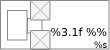
VISUALIZATION SperrAntrieb_MR_Flap_Txt_R_Below  // 110x50
VAR_INPUT
    ITF_SPERRANTRIEB_IN   	:   ITF_SPERRANTRIEB;	
END_VAR
VAR_INPUT CONSTANT
    stExklParameter		:   STRING[40] := ' ';	
END_VAR
VAR CONSTANT
	uiIconNr				:	UINT := 7;
END_VAR
    Frame (0,0 110x50), invisible if: NOT fcCheckQuerryReturnIcon(_ITF_In := ITF_SPERRANTRIEB_IN,_uiIconNr_In := uiIconNr)
        shows SperrAntrieb_MR_Flap_RB_CheckQuerry(ITF_SPERRANTRIEB_IN := ITF_SPERRANTRIEB_IN, stExklParameter := stExklParameter)
        shows Icon()
END_VISUALIZATION

// 40 Visualizations/ICON/SperrAntrieb_RIGHT/Motor_Right/Below/SperrAntrieb_MR_Flap_RB_CheckQuerry
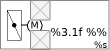
VISUALIZATION SperrAntrieb_MR_Flap_RB_CheckQuerry  // 110x50
VAR_INPUT
    ITF_SPERRANTRIEB_IN   :   ITF_SPERRANTRIEB;
    stExklParameter		:   STRING[40];	
END_VAR
    Frame (0,0 110x50)
        shows SperrAntrieb_MR_Flap_RB_CheckEnabled(ITF_SPERRANTRIEB_IN := ITF_SPERRANTRIEB_IN, stExklParameter := stExklParameter)
END_VISUALIZATION

// 40 Visualizations/ICON/SperrAntrieb_RIGHT/Motor_Right/Below/SperrAntrieb_MR_Flap_RB_CheckEnabled
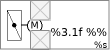
VISUALIZATION SperrAntrieb_MR_Flap_RB_CheckEnabled  // 110x50
VAR_INPUT
    ITF_SPERRANTRIEB_IN   :   ITF_SPERRANTRIEB;
    stExklParameter		:   STRING[40];	
END_VAR
    Frame (0,0 50x50), invisible if: NOT ITF_SPERRANTRIEB_IN.proIsEnabled
        shows Icon_MR_Klappe(ITF_SPERRANTRIEB_IN := ITF_SPERRANTRIEB_IN)
    Frame (50,25 60x25), invisible if: NOT ITF_SPERRANTRIEB_IN.proIsEnabled
        shows ValueDwnUp(ITF_SPERRANTRIEB_IN := ITF_SPERRANTRIEB_IN, uiTextAusrichtung := 4)
    Rectangle (0,0 110x50)
        OnMouseClick:  Dialog=SperrAntrieb_POPUP, Parameters={stExklParameter: , ITF_SPERRANTRIEBIN: ITF_SPERRANTRIEB_IN, uiPopUpGruppe: 0}, OpenCentered=True
END_VISUALIZATION

// 40 Visualizations/ICON/SperrAntrieb_BASE/Ventile/Klappe/Motor_Below/MB_Klappe_AUF
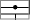
VISUALIZATION MB_Klappe_AUF  // 30x20
    Rectangle (0,0 30x14)
    Line (15,14) (15,20)
    Line (0,7) (30,7)
    Ellipse (13,5 4x4)
END_VISUALIZATION

// 40 Visualizations/ICON/SperrAntrieb_BASE/Ventile/Klappe/Motor_Left/ML_Klappe_AUF
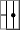
VISUALIZATION ML_Klappe_AUF  // 20x30
    Rectangle (6,0 14x30)
    Ellipse (11,13 4x4)
    Line (13,0) (13,30)
    Line (6,15) (0,15)
END_VISUALIZATION

// 40 Visualizations/ICON/SperrAntrieb_BASE/Ventile/Klappe/Motor_Right/MR_Klappe_AUF
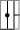
VISUALIZATION MR_Klappe_AUF  // 20x30
    Line (20,15) (14,15)
    Rectangle (0,0 14x30)
    Ellipse (5,13 4x4)
    Line (7,0) (7,30)
END_VISUALIZATION

// 40 Visualizations/ICON/SperrAntrieb_LEFT/Motor_Below/SperrAntrieb_MB_Flap_LB_CheckEnabled
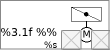
VISUALIZATION SperrAntrieb_MB_Flap_LB_CheckEnabled  // 110x50
VAR_INPUT
    ITF_SPERRANTRIEB_IN   :   ITF_SPERRANTRIEB;	
    stExklParameter		:   STRING[40];	
END_VAR
    Frame (61,0 50x50), invisible if: NOT ITF_SPERRANTRIEB_IN.proIsEnabled
        shows Icon_MB_Klappe(ITF_SPERRANTRIEB_IN := ITF_SPERRANTRIEB_IN)
    Frame (0,25 60x25), invisible if: NOT ITF_SPERRANTRIEB_IN.proIsEnabled
        shows ValueDwnUp(ITF_SPERRANTRIEB_IN := ITF_SPERRANTRIEB_IN, uiTextAusrichtung := 6)
    Rectangle (0,0 110x50)
        OnMouseClick:  Dialog=SperrAntrieb_POPUP, Parameters={stExklParameter: stExklParameter, ITF_SPERRANTRIEBIN: ITF_SPERRANTRIEB_IN, uiPopUpGruppe: 0}, OpenCentered=True
END_VISUALIZATION

// 40 Visualizations/ICON/SperrAntrieb_LEFT/Motor_Below/SperrAntrieb_MB_Flap_LB_CheckQuerry
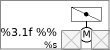
VISUALIZATION SperrAntrieb_MB_Flap_LB_CheckQuerry  // 110x50
VAR_INPUT
    ITF_SPERRANTRIEB_IN   :   ITF_SPERRANTRIEB;
    stExklParameter		:   STRING[40];	
END_VAR
    Frame (0,0 110x50)
        shows SperrAntrieb_MB_Flap_LB_CheckEnabled(ITF_SPERRANTRIEB_IN := ITF_SPERRANTRIEB_IN, stExklParameter := stExklParameter)
END_VISUALIZATION

// 40 Visualizations/ICON/SperrAntrieb_LEFT/Motor_Below/SperrAntrieb_MB_Flap_Txt_L_Below
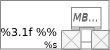
VISUALIZATION SperrAntrieb_MB_Flap_Txt_L_Below  // 110x50
VAR_INPUT
    ITF_SPERRANTRIEB_IN		:   ITF_SPERRANTRIEB;	
END_VAR
VAR_INPUT CONSTANT
    stExklParameter		:   STRING[40] := ' ';	
END_VAR
VAR CONSTANT
	uiIconNr				:	UINT := 1;
END_VAR
    Frame (0,0 110x50), invisible if: NOT fcCheckQuerryReturnIcon(_ITF_In := ITF_SPERRANTRIEB_IN,_uiIconNr_In := uiIconNr)
        shows SperrAntrieb_MB_Flap_LB_CheckQuerry(ITF_SPERRANTRIEB_IN := ITF_SPERRANTRIEB_IN, stExklParameter := stExklParameter)
        shows Icon()
END_VISUALIZATION

// 40 Visualizations/ICON/SperrAntrieb_LEFT/Motor_LEFT/Above/SperrAntrieb_ML_Flap_Txt_L_Above
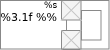
VISUALIZATION SperrAntrieb_ML_Flap_Txt_L_Above  // 110x50
VAR_INPUT
    ITF_SPERRANTRIEB_IN		:   ITF_SPERRANTRIEB;	
END_VAR
VAR_INPUT CONSTANT
    stExklParameter		:   STRING[40] := ' ';	
END_VAR
VAR CONSTANT
	uiIconNr				:	UINT := 2;
END_VAR
    Frame (0,0 110x50), invisible if: NOT fcCheckQuerryReturnIcon(_ITF_In := ITF_SPERRANTRIEB_IN,_uiIconNr_In := uiIconNr)
        shows SperrAntrieb_ML_Flap_LA_CheckQuerry(ITF_SPERRANTRIEB_IN := ITF_SPERRANTRIEB_IN, stExklParameter := stExklParameter)
        shows S_AT_ML_Valve_AB_Up_LA_CheckQuerry()
END_VISUALIZATION

// 40 Visualizations/ICON/SperrAntrieb_LEFT/Motor_LEFT/Above/SperrAntrieb_ML_Flap_LA_CheckQuerry
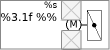
VISUALIZATION SperrAntrieb_ML_Flap_LA_CheckQuerry  // 110x50
VAR_INPUT
    ITF_SPERRANTRIEB_IN   :   ITF_SPERRANTRIEB;
    stExklParameter		:   STRING[40];	
END_VAR
    Frame (0,0 110x50)
        shows SperrAntrieb_ML_Flap_LA_CheckEnabled(ITF_SPERRANTRIEB_IN := ITF_SPERRANTRIEB_IN, stExklParameter := stExklParameter)
END_VISUALIZATION

// 40 Visualizations/ICON/SperrAntrieb_LEFT/Motor_LEFT/Above/SperrAntrieb_ML_Flap_LA_CheckEnabled
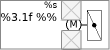
VISUALIZATION SperrAntrieb_ML_Flap_LA_CheckEnabled  // 110x50
VAR_INPUT
    ITF_SPERRANTRIEB_IN   :   ITF_SPERRANTRIEB;
    stExklParameter		:   STRING[40];	
END_VAR
    Frame (61,0 50x50), invisible if: NOT ITF_SPERRANTRIEB_IN.proIsEnabled
        shows Icon_ML_Klappe(ITF_SPERRANTRIEB_IN := ITF_SPERRANTRIEB_IN)
    Frame (0,0 60x25), invisible if: NOT ITF_SPERRANTRIEB_IN.proIsEnabled
        shows ValueUpDwn(ITF_SPERRANTRIEB_IN := ITF_SPERRANTRIEB_IN, uiTextAusrichtung := 6)
    Rectangle (0,0 110x50)
        OnMouseClick:  Dialog=SperrAntrieb_POPUP, Parameters={stExklParameter: stExklParameter, ITF_SPERRANTRIEBIN: ITF_SPERRANTRIEB_IN, uiPopUpGruppe: 0}, OpenCentered=True
END_VISUALIZATION

// 40 Visualizations/ICON/SperrAntrieb_LEFT/Motor_LEFT/Below/SperrAntrieb_ML_Flap_Txt_L_Below
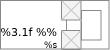
VISUALIZATION SperrAntrieb_ML_Flap_Txt_L_Below  // 110x50
VAR_INPUT
    ITF_SPERRANTRIEB_IN		:   ITF_SPERRANTRIEB;	
END_VAR
VAR_INPUT CONSTANT
    stExklParameter		:   STRING[40] := ' ';	
END_VAR
VAR CONSTANT
	uiIconNr				:	UINT := 3;
END_VAR
    Frame (0,0 110x50), invisible if: NOT fcCheckQuerryReturnIcon(_ITF_In := ITF_SPERRANTRIEB_IN,_uiIconNr_In := uiIconNr)
        shows SperrAntrieb_ML_Flap_LB_CheckQuerry(ITF_SPERRANTRIEB_IN := ITF_SPERRANTRIEB_IN, stExklParameter := stExklParameter)
        shows Icon()
END_VISUALIZATION

// 40 Visualizations/ICON/SperrAntrieb_LEFT/Motor_LEFT/Below/SperrAntrieb_ML_Flap_LB_CheckQuerry
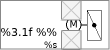
VISUALIZATION SperrAntrieb_ML_Flap_LB_CheckQuerry  // 110x50
VAR_INPUT
    ITF_SPERRANTRIEB_IN   :   ITF_SPERRANTRIEB;
    stExklParameter		:   STRING[40];	
END_VAR
    Frame (0,0 110x50)
        shows SperrAntrieb_ML_Flap_LB_CheckEnabled(ITF_SPERRANTRIEB_IN := ITF_SPERRANTRIEB_IN, stExklParameter := stExklParameter)
END_VISUALIZATION

// 40 Visualizations/ICON/SperrAntrieb_LEFT/Motor_LEFT/Below/SperrAntrieb_ML_Flap_LB_CheckEnabled
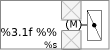
VISUALIZATION SperrAntrieb_ML_Flap_LB_CheckEnabled  // 110x50
VAR_INPUT
    ITF_SPERRANTRIEB_IN   :   ITF_SPERRANTRIEB;
    stExklParameter		:   STRING[40];	
END_VAR
    Frame (61,0 50x50), invisible if: NOT ITF_SPERRANTRIEB_IN.proIsEnabled
        shows Icon_ML_Klappe(ITF_SPERRANTRIEB_IN := ITF_SPERRANTRIEB_IN)
    Frame (0,25 60x25), invisible if: NOT ITF_SPERRANTRIEB_IN.proIsEnabled
        shows ValueDwnUp(ITF_SPERRANTRIEB_IN := ITF_SPERRANTRIEB_IN, uiTextAusrichtung := 6)
    Rectangle (0,0 110x50)
        OnMouseClick:  Dialog=SperrAntrieb_POPUP, Parameters={stExklParameter: , ITF_SPERRANTRIEBIN: ITF_SPERRANTRIEB_IN, uiPopUpGruppe: 0}, OpenCentered=True
END_VISUALIZATION

// 40 Visualizations/POPUP/PARAMETER/SperrAntrieb_Icon_SperrAntrieb
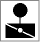
VISUALIZATION SperrAntrieb_Icon_SperrAntrieb  // 40x42
    Ellipse (13,3 14x14)
    Polygon (5,38) (5,24) (35,38)
    Polygon (5,23) (35,37) (35,23)
    Ellipse (17,27 6x6)
    Line (20,24) (20,17)
END_VISUALIZATION

// 40 Visualizations/ICON/SperrAntrieb_BASE/Value/ValueUpDwn
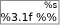
VISUALIZATION ValueUpDwn  // 60x25
VAR_INPUT
    ITF_SPERRANTRIEB_IN   :   ITF_SPERRANTRIEB;	
END_VAR
VAR_INPUT CONSTANT
    uiTextAusrichtung   : UINT := 4;    // 0 = Oben links | 1 = Horizontal zentriert | 2 = Rechts | 4 = Vertikal zentriert | 8 = Unten
END_VAR
    Textfield (0,0 60x10), "%s", text variable: ITF_SPERRANTRIEB_IN.proGetBMK, invisible if: ITF_SPERRANTRIEB_IN.proNoBmkInList
        p3718999670: uiTextAusrichtung
    Textfield (0,10 60x15), "%3.1f %%", text variable: ITF_SPERRANTRIEB_IN.proOnY, invisible if: ITF_SPERRANTRIEB_IN.proNotShowAI_ActualPosition OR NOT ITF_SPERRANTRIEB_IN.proNotShowDI_RükIsClosed OR NOT ITF_SPERRANTRIEB_IN.proNotShowDI_RükIsOpen
        p3718999670: uiTextAusrichtung
    Textfield (0,10 60x15), invisible if: NOT ITF_SPERRANTRIEB_IN.proNotShowAI_ActualPosition, text list: 'KlappenStatus', text index: ITF_SPERRANTRIEB_IN.proKlappenStatus
        p3718999670: uiTextAusrichtung
END_VISUALIZATION

// 40 Visualizations/POPUP/PARAMETER/SperrAntrieb_POPUP_IO_ITF
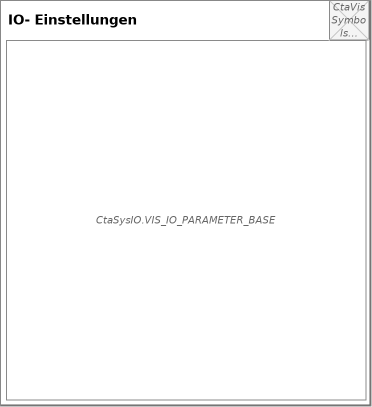
VISUALIZATION SperrAntrieb_POPUP_IO_ITF  // 372x407
VAR_INPUT
    ITF_IO_IN    :   CtaSysIO.ITF_IO;	
END_VAR
    RoundedRectangle (0,0 370x405)
    Frame (6,40 360x360)
        shows CtaSysIO.VIS_IO_PARAMETER_BASE(ITF_IO_IN := ITF_IO_IN)
        shows VIS_ANTRIEB_PARAMETER_IO1(ITF_ANTRIEBIN := ITF_ANTRIEBIN)
        shows VIS_ANTRIEB_PARAMETER_IO2(ITF_ANTRIEBIN := ITF_ANTRIEBIN)
        shows VIS_ANTRIEB_PARAMETER_IO3(ITF_ANTRIEBIN := ITF_ANTRIEBIN)
    Image (329,0 40x40), image: CtaVisSymbols.ImagePool.close_solo_black
        OnMouseClick:  Dialog=SperrAntrieb_POPUP_IO_ITF, Result=None, NumpadKeypadSet=True
    Label (5,0 150x40), "IO- Einstellungen"
END_VISUALIZATION

// 40 Visualizations/POPUP/PARAMETER/SperrAntrieb_IO/SperrAntrieb_ParameterIO4
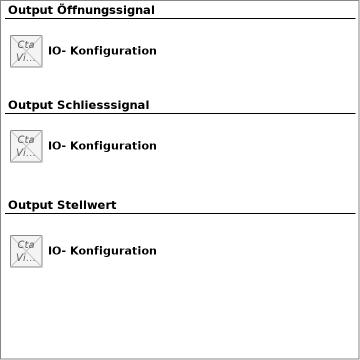
VISUALIZATION SperrAntrieb_ParameterIO4  // 360x360
VAR_INPUT
    ITF_SPERRANTRIEBIN  :   ITF_SPERRANTRIEB;	
	ITF_xOnAuf_IN		:	CtaSysIO.ITF_IO;
	ITF_xOnZu_IN		:	CtaSysIO.ITF_IO;
	ITF_rOnY_IN			:	CtaSysIO.ITF_IO;
END_VAR
    Label (5,0 350x20), "Output Öffnungssignal"
    Label (5,195 350x20), "Output Stellwert"
    Line (5,213) (355,213)
    Line (5,18) (355,18)
    Image (10,35 32x32), invisible if: ITF_xOnAuf_IN = 0, image: CtaVisSymbols.ImagePool.build
        OnMouseDown:  Dialog=SperrAntrieb_POPUP_IO_ITF, Parameters={ITF_IO_IN: ITF_xOnAuf_IN}, OpenModal=True, OpenCentered=True
    Image (10,235 32x32), invisible if: ITF_rOnY_IN = 0, image: CtaVisSymbols.ImagePool.build
        OnMouseDown:  Dialog=SperrAntrieb_POPUP_IO_ITF, Parameters={ITF_IO_IN: ITF_rOnY_IN}, OpenModal=True, OpenCentered=True
    Label (45,41 120x20), "IO- Konfiguration", invisible if: ITF_xOnAuf_IN = 0
    Label (45,241 120x20), "IO- Konfiguration", invisible if: ITF_rOnY_IN = 0
    Line (5,113) (355,113)
    Label (5,95 350x20), "Output Schliesssignal"
    Image (10,130 32x32), invisible if: ITF_xOnZu_IN = 0, image: CtaVisSymbols.ImagePool.build
        OnMouseDown:  Dialog=SperrAntrieb_POPUP_IO_ITF, Parameters={ITF_IO_IN: ITF_xOnZu_IN}, OpenModal=True, OpenCentered=True
    Label (45,136 120x20), "IO- Konfiguration", invisible if: ITF_xOnZu_IN = 0
END_VISUALIZATION

// 40 Visualizations/ICON/SperrAntrieb_BASE/Value/ValueDwnUp
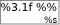
VISUALIZATION ValueDwnUp  // 60x25
VAR_INPUT
    ITF_SPERRANTRIEB_IN   :   ITF_SPERRANTRIEB;	
END_VAR
VAR_INPUT CONSTANT
    uiTextAusrichtung   : UINT := 4;    // 0 = Oben links | 1 = Horizontal zentriert | 2 = Rechts | 4 = Vertikal zentriert | 8 = Unten
END_VAR
    Textfield (0,0 60x15), "%3.1f %%", text variable: ITF_SPERRANTRIEB_IN.proOnY, invisible if: ITF_SPERRANTRIEB_IN.proNotShowAI_ActualPosition OR NOT ITF_SPERRANTRIEB_IN.proNotShowDI_RükIsClosed OR NOT ITF_SPERRANTRIEB_IN.proNotShowDI_RükIsOpen
        p3718999670: uiTextAusrichtung
    Textfield (0,0 60x15), invisible if: NOT ITF_SPERRANTRIEB_IN.proNotShowAI_ActualPosition, text list: 'KlappenStatus', text index: ITF_SPERRANTRIEB_IN.proKlappenStatus
        p3718999670: uiTextAusrichtung
    Textfield (0,15 60x10), "%s", text variable: ITF_SPERRANTRIEB_IN.proGetBMK, invisible if: ITF_SPERRANTRIEB_IN.proNoBmkInList
        p3718999670: uiTextAusrichtung
END_VISUALIZATION

// 40 Visualizations/ICON/SperrAntrieb_LEFT/Motor_Right/Above/SperrAntrieb_MR_Flap_Txt_L_Above
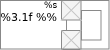
VISUALIZATION SperrAntrieb_MR_Flap_Txt_L_Above  // 110x50
VAR_INPUT
    ITF_SPERRANTRIEB_IN		:   ITF_SPERRANTRIEB;	
END_VAR
VAR_INPUT CONSTANT
    stExklParameter		:   STRING[40] := ' ';	
END_VAR
VAR CONSTANT
	uiIconNr				:	UINT := 2;
END_VAR
    Frame (0,0 110x50), invisible if: NOT fcCheckQuerryReturnIcon(_ITF_In := ITF_SPERRANTRIEB_IN,_uiIconNr_In := uiIconNr)
        shows SperrAntrieb_ML_Flap_LA_CheckQuerry(ITF_SPERRANTRIEB_IN := ITF_SPERRANTRIEB_IN, stExklParameter := stExklParameter)
        shows S_AT_ML_Valve_AB_Up_LA_CheckQuerry()
END_VISUALIZATION

// 40 Visualizations/ICON/SperrAntrieb_LEFT/Motor_Right/Above/SperrAntrieb_MR_Flap_LA_CheckQuerry
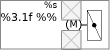
VISUALIZATION SperrAntrieb_MR_Flap_LA_CheckQuerry  // 110x50
VAR_INPUT
    ITF_SPERRANTRIEB_IN   :   ITF_SPERRANTRIEB;
    stExklParameter		:   STRING[40];	
END_VAR
    Frame (0,0 110x50)
        shows SperrAntrieb_ML_Flap_LA_CheckEnabled(ITF_SPERRANTRIEB_IN := ITF_SPERRANTRIEB_IN, stExklParameter := stExklParameter)
END_VISUALIZATION

// 40 Visualizations/ICON/SperrAntrieb_LEFT/Motor_Right/Above/SperrAntrieb_MR_Flap_LA_CheckEnabled
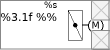
VISUALIZATION SperrAntrieb_MR_Flap_LA_CheckEnabled  // 110x50
VAR_INPUT
    ITF_SPERRANTRIEB_IN   :   ITF_SPERRANTRIEB;
    stExklParameter		:   STRING[40];	
END_VAR
    Frame (61,0 50x50), invisible if: NOT ITF_SPERRANTRIEB_IN.proIsEnabled
        shows Icon_MR_Klappe(ITF_SPERRANTRIEB_IN := ITF_SPERRANTRIEB_IN)
    Frame (0,0 60x25), invisible if: NOT ITF_SPERRANTRIEB_IN.proIsEnabled
        shows ValueUpDwn(ITF_SPERRANTRIEB_IN := ITF_SPERRANTRIEB_IN, uiTextAusrichtung := 6)
    Rectangle (0,0 110x50)
        OnMouseClick:  Dialog=SperrAntrieb_POPUP, Parameters={stExklParameter: stExklParameter, ITF_SPERRANTRIEBIN: ITF_SPERRANTRIEB_IN, uiPopUpGruppe: 0}, OpenCentered=True
END_VISUALIZATION

// 40 Visualizations/ICON/SperrAntrieb_LEFT/Motor_Right/Below/SperrAntrieb_MR_Flap_Txt_L_Below
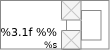
VISUALIZATION SperrAntrieb_MR_Flap_Txt_L_Below  // 110x50
VAR_INPUT
    ITF_SPERRANTRIEB_IN		:   ITF_SPERRANTRIEB;	
END_VAR
VAR_INPUT CONSTANT
    stExklParameter		:   STRING[40] := ' ';	
END_VAR
VAR CONSTANT
	uiIconNr				:	UINT := 3;
END_VAR
    Frame (0,0 110x50), invisible if: NOT fcCheckQuerryReturnIcon(_ITF_In := ITF_SPERRANTRIEB_IN,_uiIconNr_In := uiIconNr)
        shows SperrAntrieb_ML_Flap_LB_CheckQuerry(ITF_SPERRANTRIEB_IN := ITF_SPERRANTRIEB_IN, stExklParameter := stExklParameter)
        shows Icon()
END_VISUALIZATION

// 40 Visualizations/ICON/SperrAntrieb_LEFT/Motor_Right/Below/SperrAntrieb_MR_Flap_LB_CheckQuerry
